(* CODESYS project bibliothek.library
   Company: er
   Title: er
   Placeholder: er
   Version: 0.0.1

Project tree, tasks and I/O mapping:
  libraries: GWP Library, * (Viessmann); Tc2_Standard, * (Beckhoff Automation GmbH); Tc2_System, * (Beckhoff Automation GmbH); Tc2_Utilities, * (Beckhoff Automation GmbH); Tc3_Module, * (Beckhoff Automation GmbH); VisuDialogs, * (System)
  DUTs/
    GVLs/
      global variables Globale_Uhr
  POUs/
    Funktionsblock/
    program MAIN [ST]
    program test [FBD]
  Version/
    global variables Global_Version
  VISUs/
    Alarmliste/
      visualisation Alarmliste
    Anlageseite_6/
      visualisation Kaeltekreis6_1
      visualisation Sollwertaenderung_C_6_3
      visualisation Zustandsanzeige
    Hauptmenu_3/
      visualisation Fusszeile_50
      visualisation Hauptmenu
      visualisation Kontaktseite3_1_50
      visualisation Uhr_einstellen3_1_50
    Home/
      visualisation Auswahlmenue
      visualisation Ein_Aus_Schalter
      visualisation Home_Standard_50
      visualisation RI_Schema_50
    IBN/
      visualisation IO_Auswahl
      visualisation Liste_AO
      visualisation Liste_DI
      visualisation SW_IBN_Einstellungen_K
    Infoseite/
      visualisation Infoliste
      visualisation Infoseite
    Sollwertmenu_9/
      Sollwertmenu/
        visualisation Sollwertmenu
      Wärmegewinnung/
        UWP/
          visualisation SW_Einstellungen_C
          visualisation SW_Einstellungen_DT
          visualisation SW_Einstellungen_K
          visualisation SW_Einstellungen_Zeit
          visualisation SW_WG_UWP_Verd
          visualisation SW_WG_UWP_Verd_Liste
        visualisation Sollwertmenu_Waermegewinnung
      Wärmepumpe/
      Wärmesenke/
      visualisation _SW_Heizgruppe
      visualisation _SW_Speicher_BWW
      visualisation _SW_Speicher_Heizung_1
      visualisation _SW_Speicher_Kaltwasser
      visualisation _SW_Waermegewinnung
      visualisation Sollwertmenu_Waermesenke
      visualisation SW_Waermepumpe
    Zeitprogramm/
      visualisation Wochenuhr_W7
    image pool Icon
    text list Sprachen
    visualisation test_1
  00000000-0000-0000-0000-000000000000|C:\Users\kuzr\Documents\Visual Studio 2013\Bildersammlung_VI\IC_102000\energietraeger_biomasse_fehler.png
  00000000-0000-0000-0000-000000000000|C:\Users\kuzr\Documents\Visual Studio 2013\Bildersammlung_VI\IC_102000\energietraeger_biomasse_inaktiv.png
  00000000-0000-0000-0000-000000000000|C:\Users\kuzr\Documents\Visual Studio 2013\Bildersammlung_VI\IC_102000\energietraeger_gas.png
  00000000-0000-0000-0000-000000000000|C:\Users\kuzr\Documents\Visual Studio 2013\Bildersammlung_VI\IC_102000\energietraeger_gas_fehler.png
  00000000-0000-0000-0000-000000000000|C:\Users\kuzr\Documents\Visual Studio 2013\Bildersammlung_VI\IC_102000\energietraeger_naturwaerme.png
  00000000-0000-0000-0000-000000000000|C:\Users\kuzr\Documents\Visual Studio 2013\Bildersammlung_VI\IC_102000\energietraeger_naturwaerme_fehler (2).png
  00000000-0000-0000-0000-000000000000|C:\Users\kuzr\Documents\Visual Studio 2013\Bildersammlung_VI\IC_102000\energietraeger_naturwaerme_fehler.png
  00000000-0000-0000-0000-000000000000|C:\Users\kuzr\Documents\Visual Studio 2013\Bildersammlung_VI\IC_102000\energietraeger_naturwaerme_inaktiv.png
  00000000-0000-0000-0000-000000000000|C:\Users\kuzr\Documents\Visual Studio 2013\Bildersammlung_VI\IC_102000\energietraeger_oel.png
  00000000-0000-0000-0000-000000000000|C:\Users\kuzr\Documents\Visual Studio 2013\Bildersammlung_VI\IC_102000\energietraeger_oel_inaktiv.png
  00000000-0000-0000-0000-000000000000|C:\Users\kuzr\Documents\Visual Studio 2013\Bildersammlung_VI\IC_102000\heizkreis_direkt (2).png
  00000000-0000-0000-0000-000000000000|C:\Users\kuzr\Documents\Visual Studio 2013\Bildersammlung_VI\IC_102000\heizkreis_direkt.png
  00000000-0000-0000-0000-000000000000|C:\Users\kuzr\Documents\Visual Studio 2013\Bildersammlung_VI\IC_102000\heizkreis_direkt_fehler.png
  00000000-0000-0000-0000-000000000000|C:\Users\kuzr\Documents\Visual Studio 2013\Bildersammlung_VI\IC_102000\heizkreis_direkt_inaktiv (2).png
  00000000-0000-0000-0000-000000000000|C:\Users\kuzr\Documents\Visual Studio 2013\Bildersammlung_VI\IC_102000\heizkreis_direkt_inaktiv.png
  00000000-0000-0000-0000-000000000000|C:\Users\kuzr\Documents\Visual Studio 2013\Bildersammlung_VI\IC_102000\heizkreis_fussbodenheizung.png
  00000000-0000-0000-0000-000000000000|C:\Users\kuzr\Documents\Visual Studio 2013\Bildersammlung_VI\IC_102000\heizkreis_fussbodenheizung_fehler.png
  00000000-0000-0000-0000-000000000000|C:\Users\kuzr\Documents\Visual Studio 2013\Bildersammlung_VI\IC_102000\heizkreis_fussbodenheizung_inaktiv.png
  00000000-0000-0000-0000-000000000000|C:\Users\kuzr\Documents\Visual Studio 2013\Bildersammlung_VI\IC_102000\heizkreis_mischer.png
  00000000-0000-0000-0000-000000000000|C:\Users\kuzr\Documents\Visual Studio 2013\Bildersammlung_VI\IC_102000\heizkreis_mischer_fehler.png
  00000000-0000-0000-0000-000000000000|C:\Users\kuzr\Documents\Visual Studio 2013\Bildersammlung_VI\IC_102000\heizkreis_mischer_inaktiv.png
  00000000-0000-0000-0000-000000000000|C:\Users\kuzr\Documents\Visual Studio 2013\Bildersammlung_VI\IC_102000\IC_102015_klappen_02.png
  00000000-0000-0000-0000-000000000000|C:\Users\kuzr\Documents\Visual Studio 2013\Bildersammlung_VI\IC_102000\klappen_01 (2).png
  00000000-0000-0000-0000-000000000000|C:\Users\kuzr\Documents\Visual Studio 2013\Bildersammlung_VI\IC_102000\klappen_01.png
  00000000-0000-0000-0000-000000000000|C:\Users\kuzr\Documents\Visual Studio 2013\Bildersammlung_VI\IC_102000\klappen_02.png
  00000000-0000-0000-0000-000000000000|C:\Users\kuzr\Documents\Visual Studio 2013\Bildersammlung_VI\IC_102000\komponente_detail_heizkreis.png
  00000000-0000-0000-0000-000000000000|C:\Users\kuzr\Documents\Visual Studio 2013\Bildersammlung_VI\IC_102000\komponente_detail_klappe (2).png
  00000000-0000-0000-0000-000000000000|C:\Users\kuzr\Documents\Visual Studio 2013\Bildersammlung_VI\IC_102000\komponente_detail_klappe.png
  00000000-0000-0000-0000-000000000000|C:\Users\kuzr\Documents\Visual Studio 2013\Bildersammlung_VI\IC_102000\komponente_detail_klappe_fehler (2).png
  00000000-0000-0000-0000-000000000000|C:\Users\kuzr\Documents\Visual Studio 2013\Bildersammlung_VI\IC_102000\komponente_detail_klappe_fehler.png
  00000000-0000-0000-0000-000000000000|C:\Users\kuzr\Documents\Visual Studio 2013\Bildersammlung_VI\IC_102000\komponente_detail_klappe_inaktiv.png
  00000000-0000-0000-0000-000000000000|C:\Users\kuzr\Documents\Visual Studio 2013\Bildersammlung_VI\IC_102000\komponente_detail_klappe_inaktiv_2.png
  00000000-0000-0000-0000-000000000000|C:\Users\kuzr\Documents\Visual Studio 2013\Bildersammlung_VI\IC_102000\komponente_detail_mischer_01.png
  00000000-0000-0000-0000-000000000000|C:\Users\kuzr\Documents\Visual Studio 2013\Bildersammlung_VI\IC_102000\komponente_detail_mischer_02.png
  00000000-0000-0000-0000-000000000000|C:\Users\kuzr\Documents\Visual Studio 2013\Bildersammlung_VI\IC_102000\komponente_detail_mischer_fehler.png
  00000000-0000-0000-0000-000000000000|C:\Users\kuzr\Documents\Visual Studio 2013\Bildersammlung_VI\IC_102000\komponente_detail_mischer_inaktiv.png
  00000000-0000-0000-0000-000000000000|C:\Users\kuzr\Documents\Visual Studio 2013\Bildersammlung_VI\IC_102000\komponente_detail_pumpe.png
  00000000-0000-0000-0000-000000000000|C:\Users\kuzr\Documents\Visual Studio 2013\Bildersammlung_VI\IC_102000\komponente_detail_pumpe_fehler.png
  00000000-0000-0000-0000-000000000000|C:\Users\kuzr\Documents\Visual Studio 2013\Bildersammlung_VI\IC_102000\komponente_detail_pumpe_inaktiv.png
  00000000-0000-0000-0000-000000000000|C:\Users\kuzr\Documents\Visual Studio 2013\Bildersammlung_VI\IC_102000\mischer_01.png
  00000000-0000-0000-0000-000000000000|C:\Users\kuzr\Documents\Visual Studio 2013\Bildersammlung_VI\IC_102000\mischer_02.png
  00000000-0000-0000-0000-000000000000|C:\Users\kuzr\Documents\Visual Studio 2013\Bildersammlung_VI\IC_102000\mischer_03.png
  00000000-0000-0000-0000-000000000000|C:\Users\kuzr\Documents\Visual Studio 2013\Bildersammlung_VI\IC_102000\mischer_04.png
  00000000-0000-0000-0000-000000000000|C:\Users\kuzr\Documents\Visual Studio 2013\Bildersammlung_VI\IC_102000\mischer_05.png
  00000000-0000-0000-0000-000000000000|C:\Users\kuzr\Documents\Visual Studio 2013\Bildersammlung_VI\IC_102000\mischer_06.png
  00000000-0000-0000-0000-000000000000|C:\Users\kuzr\Documents\Visual Studio 2013\Bildersammlung_VI\IC_102000\mischer_07.png
  00000000-0000-0000-0000-000000000000|C:\Users\kuzr\Documents\Visual Studio 2013\Bildersammlung_VI\IC_102000\mischer_08.png
  00000000-0000-0000-0000-000000000000|C:\Users\kuzr\Documents\Visual Studio 2013\Bildersammlung_VI\IC_102000\mischer_09.png
  00000000-0000-0000-0000-000000000000|C:\Users\kuzr\Documents\Visual Studio 2013\Bildersammlung_VI\IC_102000\mischer_10.png
  00000000-0000-0000-0000-000000000000|C:\Users\kuzr\Documents\Visual Studio 2013\Bildersammlung_VI\IC_102000\mischer_11.png
  00000000-0000-0000-0000-000000000000|C:\Users\kuzr\Documents\Visual Studio 2013\Bildersammlung_VI\IC_102000\mischer_12.png
  00000000-0000-0000-0000-000000000000|C:\Users\kuzr\Documents\Visual Studio 2013\Bildersammlung_VI\IC_102000\pumpe_links.png
  00000000-0000-0000-0000-000000000000|C:\Users\kuzr\Documents\Visual Studio 2013\Bildersammlung_VI\IC_102000\pumpe_oben.png
  00000000-0000-0000-0000-000000000000|C:\Users\kuzr\Documents\Visual Studio 2013\Bildersammlung_VI\IC_102000\pumpe_rechts.png
  00000000-0000-0000-0000-000000000000|C:\Users\kuzr\Documents\Visual Studio 2013\Bildersammlung_VI\IC_102000\pumpe_unten.png
  00000000-0000-0000-0000-000000000000|C:\Users\kuzr\Documents\Visual Studio 2013\Bildersammlung_VI\IC_102000\speicher_eis.png
  00000000-0000-0000-0000-000000000000|C:\Users\kuzr\Documents\Visual Studio 2013\Bildersammlung_VI\IC_102000\speicher_eis_fehler.png
  00000000-0000-0000-0000-000000000000|C:\Users\kuzr\Documents\Visual Studio 2013\Bildersammlung_VI\IC_102000\speicher_eis_inaktiv.png
  00000000-0000-0000-0000-000000000000|C:\Users\kuzr\Documents\Visual Studio 2013\Bildersammlung_VI\IC_102000\speicher_heizen.png
  00000000-0000-0000-0000-000000000000|C:\Users\kuzr\Documents\Visual Studio 2013\Bildersammlung_VI\IC_102000\speicher_heizen_fehler.png
  00000000-0000-0000-0000-000000000000|C:\Users\kuzr\Documents\Visual Studio 2013\Bildersammlung_VI\IC_102000\speicher_heizen_inaktiv.png
  00000000-0000-0000-0000-000000000000|C:\Users\kuzr\Documents\Visual Studio 2013\Bildersammlung_VI\IC_102000\speicher_warmwasser.png
  00000000-0000-0000-0000-000000000000|C:\Users\kuzr\Documents\Visual Studio 2013\Bildersammlung_VI\IC_102000\speicher_warmwasser_fehler.png
  00000000-0000-0000-0000-000000000000|C:\Users\kuzr\Documents\Visual Studio 2013\Bildersammlung_VI\IC_102000\speicher_warmwasser_inaktiv.png
  00000000-0000-0000-0000-000000000000|C:\Users\kuzr\Documents\Visual Studio 2013\Bildersammlung_VI\IC_102000\energietraeger_biomasse.png
  00000000-0000-0000-0000-000000000000|C:\Users\kuzr\Documents\Visual Studio 2013\Bildersammlung_VI\IC_106000\komponente_brenner.png
  00000000-0000-0000-0000-000000000000|C:\Users\kuzr\Documents\Visual Studio 2013\Bildersammlung_VI\IC_106000\komponente_brenner_fehler.png
  00000000-0000-0000-0000-000000000000|C:\Users\kuzr\Documents\Visual Studio 2013\Bildersammlung_VI\IC_106000\komponente_brenner_inaktiv.png
  00000000-0000-0000-0000-000000000000|C:\Users\kuzr\Documents\Visual Studio 2013\Bildersammlung_VI\IC_106000\speicher.png
  00000000-0000-0000-0000-000000000000|C:\Users\kuzr\Documents\Visual Studio 2013\Bildersammlung_VI\IC_106000\speicher_eis.png
  00000000-0000-0000-0000-000000000000|C:\Users\kuzr\Documents\Visual Studio 2013\Bildersammlung_VI\IC_106000\system_leistung_nicht_touchbar.png
  00000000-0000-0000-0000-000000000000|C:\Users\kuzr\Documents\Visual Studio 2013\Bildersammlung_VI\IC_106000\system_leistung_touchbar.png
  00000000-0000-0000-0000-000000000000|C:\Users\kuzr\Documents\Visual Studio 2013\Bildersammlung_VI\IC_106000\waermetauscher.png
  00000000-0000-0000-0000-000000000000|C:\Users\kuzr\Documents\Visual Studio 2013\Bildersammlung_VI\IC_106000\weiche.png
  00000000-0000-0000-0000-000000000000|C:\Users\kuzr\Documents\Visual Studio 2013\Bildersammlung_VI\IC_108000\komponente_brenner_fehler.png
  00000000-0000-0000-0000-000000000000|C:\Users\kuzr\Documents\Visual Studio 2013\Bildersammlung_VI\IC_108000\komponente_brenner_inaktiv.png
  00000000-0000-0000-0000-000000000000|C:\Users\kuzr\Documents\Visual Studio 2013\Bildersammlung_VI\IC_108000\speicher.png
  00000000-0000-0000-0000-000000000000|C:\Users\kuzr\Documents\Visual Studio 2013\Bildersammlung_VI\IC_108000\speicher_eis.png
  00000000-0000-0000-0000-000000000000|C:\Users\kuzr\Documents\Visual Studio 2013\Bildersammlung_VI\IC_108000\komponente_brenner.png
  00000000-0000-0000-0000-000000000000|C:\Users\kuzr\Documents\Visual Studio 2013\Bildersammlung_VI\IC_111000\bildschirm_reinigen.png
  00000000-0000-0000-0000-000000000000|C:\Users\kuzr\Documents\Visual Studio 2013\Bildersammlung_VI\IC_111000\dokumentation.png
  00000000-0000-0000-0000-000000000000|C:\Users\kuzr\Documents\Visual Studio 2013\Bildersammlung_VI\IC_111000\kontaktdaten_nutzer.png
  00000000-0000-0000-0000-000000000000|C:\Users\kuzr\Documents\Visual Studio 2013\Bildersammlung_VI\IC_111000\kontaktdaten_viessmann.png
  00000000-0000-0000-0000-000000000000|C:\Users\kuzr\Documents\Visual Studio 2013\Bildersammlung_VI\IC_111000\nutzeranmeldung.png
  00000000-0000-0000-0000-000000000000|C:\Users\kuzr\Documents\Visual Studio 2013\Bildersammlung_VI\IC_111000\oberflaeche_schließen.png
  00000000-0000-0000-0000-000000000000|C:\Users\kuzr\Documents\Visual Studio 2013\Bildersammlung_VI\IC_111000\pruefbetrieb.png
  00000000-0000-0000-0000-000000000000|C:\Users\kuzr\Documents\Visual Studio 2013\Bildersammlung_VI\IC_111000\system_konfigurieren.png
  00000000-0000-0000-0000-000000000000|C:\Users\kuzr\Documents\Visual Studio 2013\Bildersammlung_VI\IC_111000\betriebszaehler_zuruecksetzen.png
  00000000-0000-0000-0000-000000000000|C:\Users\kuzr\Documents\Visual Studio 2013\Bildersammlung_VI\IC_112000\abschaltbetrieb.png
  00000000-0000-0000-0000-000000000000|C:\Users\kuzr\Documents\Visual Studio 2013\Bildersammlung_VI\IC_112000\aktiv.png
  00000000-0000-0000-0000-000000000000|C:\Users\kuzr\Documents\Visual Studio 2013\Bildersammlung_VI\IC_112000\an.png
  00000000-0000-0000-0000-000000000000|C:\Users\kuzr\Documents\Visual Studio 2013\Bildersammlung_VI\IC_112000\astatur_01.png
  00000000-0000-0000-0000-000000000000|C:\Users\kuzr\Documents\Visual Studio 2013\Bildersammlung_VI\IC_112000\auf.png
  00000000-0000-0000-0000-000000000000|C:\Users\kuzr\Documents\Visual Studio 2013\Bildersammlung_VI\IC_112000\aus.png
  00000000-0000-0000-0000-000000000000|C:\Users\kuzr\Documents\Visual Studio 2013\Bildersammlung_VI\IC_112000\bedingung_erfuellt.png
  00000000-0000-0000-0000-000000000000|C:\Users\kuzr\Documents\Visual Studio 2013\Bildersammlung_VI\IC_112000\bedingung_nicht_erfuellt.png
  00000000-0000-0000-0000-000000000000|C:\Users\kuzr\Documents\Visual Studio 2013\Bildersammlung_VI\IC_112000\email_prueftaste.png
  00000000-0000-0000-0000-000000000000|C:\Users\kuzr\Documents\Visual Studio 2013\Bildersammlung_VI\IC_112000\erfuellt.png
  00000000-0000-0000-0000-000000000000|C:\Users\kuzr\Documents\Visual Studio 2013\Bildersammlung_VI\IC_112000\exportieren.png
  00000000-0000-0000-0000-000000000000|C:\Users\kuzr\Documents\Visual Studio 2013\Bildersammlung_VI\IC_112000\frostschutzbetrieb.png
  00000000-0000-0000-0000-000000000000|C:\Users\kuzr\Documents\Visual Studio 2013\Bildersammlung_VI\IC_112000\haeckchen_ungesetzt (2).png
  00000000-0000-0000-0000-000000000000|C:\Users\kuzr\Documents\Visual Studio 2013\Bildersammlung_VI\IC_112000\haeckchen_ungesetzt.png
  00000000-0000-0000-0000-000000000000|C:\Users\kuzr\Documents\Visual Studio 2013\Bildersammlung_VI\IC_112000\home.png
  00000000-0000-0000-0000-000000000000|C:\Users\kuzr\Documents\Visual Studio 2013\Bildersammlung_VI\IC_112000\home_uebersicht.png
  00000000-0000-0000-0000-000000000000|C:\Users\kuzr\Documents\Visual Studio 2013\Bildersammlung_VI\IC_112000\inaktiv.png
  00000000-0000-0000-0000-000000000000|C:\Users\kuzr\Documents\Visual Studio 2013\Bildersammlung_VI\IC_112000\intervall.png
  00000000-0000-0000-0000-000000000000|C:\Users\kuzr\Documents\Visual Studio 2013\Bildersammlung_VI\IC_112000\Itastatur_03.png
  00000000-0000-0000-0000-000000000000|C:\Users\kuzr\Documents\Visual Studio 2013\Bildersammlung_VI\IC_112000\ja.png
  00000000-0000-0000-0000-000000000000|C:\Users\kuzr\Documents\Visual Studio 2013\Bildersammlung_VI\IC_112000\kopieren.png
  00000000-0000-0000-0000-000000000000|C:\Users\kuzr\Documents\Visual Studio 2013\Bildersammlung_VI\IC_112000\laden.png
  00000000-0000-0000-0000-000000000000|C:\Users\kuzr\Documents\Visual Studio 2013\Bildersammlung_VI\IC_112000\listenansicht.png
  00000000-0000-0000-0000-000000000000|C:\Users\kuzr\Documents\Visual Studio 2013\Bildersammlung_VI\IC_112000\meldelisten_archiv.png
  00000000-0000-0000-0000-000000000000|C:\Users\kuzr\Documents\Visual Studio 2013\Bildersammlung_VI\IC_112000\meldelisten_einstellungen.png
  00000000-0000-0000-0000-000000000000|C:\Users\kuzr\Documents\Visual Studio 2013\Bildersammlung_VI\IC_112000\meldungen_weiterleiten.png
  00000000-0000-0000-0000-000000000000|C:\Users\kuzr\Documents\Visual Studio 2013\Bildersammlung_VI\IC_112000\menue.png
  00000000-0000-0000-0000-000000000000|C:\Users\kuzr\Documents\Visual Studio 2013\Bildersammlung_VI\IC_112000\minus.png
  00000000-0000-0000-0000-000000000000|C:\Users\kuzr\Documents\Visual Studio 2013\Bildersammlung_VI\IC_112000\nein.png
  00000000-0000-0000-0000-000000000000|C:\Users\kuzr\Documents\Visual Studio 2013\Bildersammlung_VI\IC_112000\nicht_erfuellt.png
  00000000-0000-0000-0000-000000000000|C:\Users\kuzr\Documents\Visual Studio 2013\Bildersammlung_VI\IC_112000\normalbetrieb.png
  00000000-0000-0000-0000-000000000000|C:\Users\kuzr\Documents\Visual Studio 2013\Bildersammlung_VI\IC_112000\pfeil_rechts.png
  00000000-0000-0000-0000-000000000000|C:\Users\kuzr\Documents\Visual Studio 2013\Bildersammlung_VI\IC_112000\plus.png
  00000000-0000-0000-0000-000000000000|C:\Users\kuzr\Documents\Visual Studio 2013\Bildersammlung_VI\IC_112000\quittieren_aus.png
  00000000-0000-0000-0000-000000000000|C:\Users\kuzr\Documents\Visual Studio 2013\Bildersammlung_VI\IC_112000\quittierena_an.png
  00000000-0000-0000-0000-000000000000|C:\Users\kuzr\Documents\Visual Studio 2013\Bildersammlung_VI\IC_112000\radiobutton_gesetzt.png
  00000000-0000-0000-0000-000000000000|C:\Users\kuzr\Documents\Visual Studio 2013\Bildersammlung_VI\IC_112000\radiobutton_ungesetzt.png
  text list GlobalTextList
*)

// DUTs/GVLs/Globale_Uhr
{attribute 'qualified_only'}
VAR_GLOBAL
	
	   systemtimestruct		: timestruct;   
END_VAR

// Version/Global_Version
{attribute 'TcGenerated'}
// This function has been automatically generated from the project information.
VAR_GLOBAL CONSTANT
	{attribute 'const_non_replaced'}
	{attribute 'linkalways'}
	stLibVersion_er : ST_LibVersion := (iMajor := 0, iMinor := 0, iBuild := 1, iRevision := 0, sVersion := '0.0.1');
END_VAR

// POUs/MAIN
PROGRAM MAIN
VAR

	

END_VAR

END_PROGRAM

// POUs/test
PROGRAM test
VAR

	
	Globale_Zeit_0: Globale_Zeit;
    CLK_W_0: CLK_W;
	
	GR_2_0: GR_2;
	
	


	CLK_W7_0: CLK_W7;
	Logger_0: Logger;
	GR_4_mit_RE_0: GR_4_mit_RE;
END_VAR

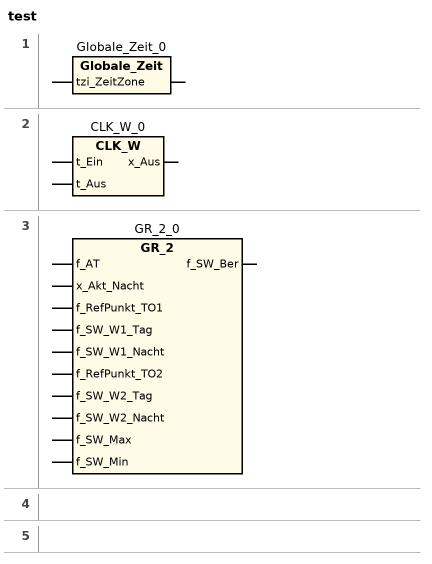
// NETWORK 1
Globale_Zeit_0(); // Globale_Zeit

// NETWORK 2
CLK_W_0(); // CLK_W

// NETWORK 3
GR_2_0(); // GR_2

// NETWORK 4

// NETWORK 5

END_PROGRAM

// VISUs/Alarmliste/Alarmliste
VISUALIZATION Alarmliste  // 800x430
END_VISUALIZATION

// VISUs/Anlageseite_6/Kaeltekreis6_1
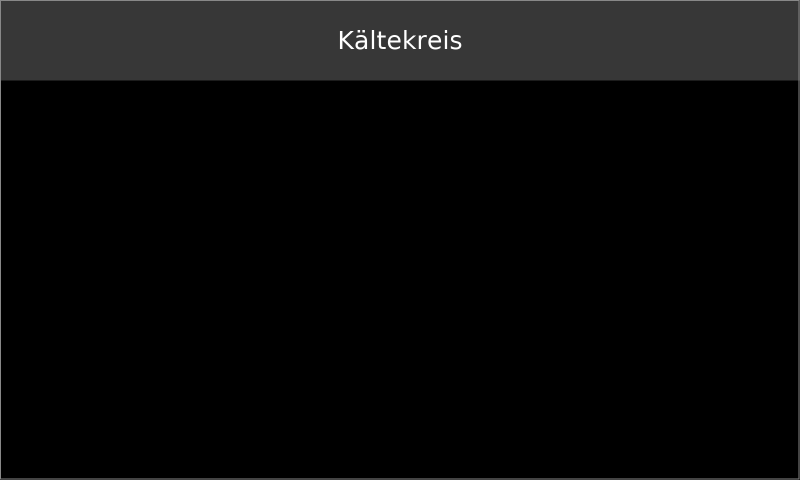
VISUALIZATION Kaeltekreis6_1  // 800x480
    Rectangle (0,0 800x80), "Kältekreis"
END_VISUALIZATION

// VISUs/Anlageseite_6/Sollwertaenderung_C_6_3
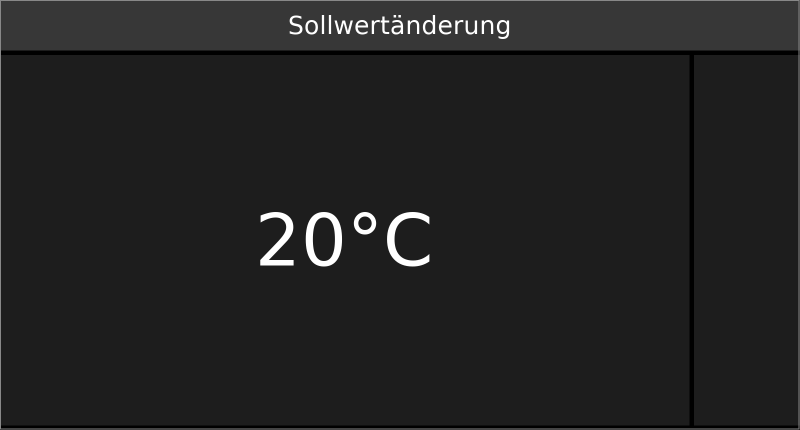
VISUALIZATION Sollwertaenderung_C_6_3  // 800x430
    Rectangle (0,0 800x50), "Sollwertänderung"
    Rectangle (0,55 689x370), "20°C"
    Rectangle (694,55 106x370)
END_VISUALIZATION

// VISUs/Anlageseite_6/Zustandsanzeige
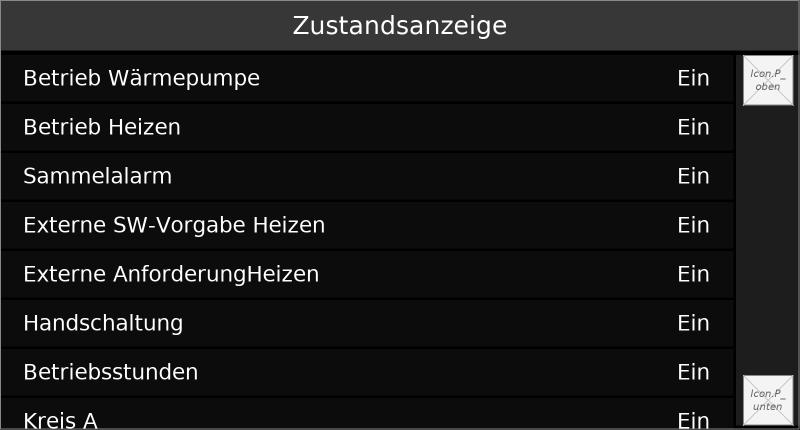
VISUALIZATION Zustandsanzeige  // 800x430
VAR_IN_OUT
	auf:BOOL;
		
END_VAR
    Image (1113,281 30x116), image: Icon.waermetauscher
    Group (0,0 800x640)
        Rectangle (0,0 800x50), "Zustandsanzeige"
        Group (0,430 800x50)
            Rectangle (0,0 800x50)
            Image (25,0 50x50), image: Icon.home
            Image (425,0 50x50), image: Icon.reinnavigieren
            Image (625,0 50x50), image: Icon.warnung_rot
            Image (125,0 50x50), image: Icon.zurueck
            Image (325,0 50x50), image: Icon.reinnavigieren
            Image (325,0 50x50), image: Icon.p_links
            Image (425,0 50x50), image: Icon.P_rechts
        Rectangle (0,55 733x46)
        Label (20,55 479x46), "Betrieb Wärmepumpe"
        Rectangle (0,104 733x46)
        Label (20,104 479x46), "Betrieb Heizen"
        Rectangle (0,153 733x46)
        Label (20,153 479x46), "Sammelalarm"
        Rectangle (0,202 733x46)
        Label (20,202 479x46), "Externe SW-Vorgabe Heizen"
        Rectangle (0,251 733x46)
        Label (20,251 479x46), "Externe AnforderungHeizen"
        Rectangle (0,300 733x46)
        Label (20,300 479x46), "Handschaltung"
        Rectangle (0,349 733x46)
        Label (20,349 479x46), "Betriebsstunden"
        Rectangle (583,55 130x46), "Ein"
        Rectangle (583,104 130x46), "Ein"
        Rectangle (0,398 733x46)
        Label (20,398 479x46), "Kreis A"
        Rectangle (0,447 733x46)
        Label (20,447 479x46), "Kreis B"
        Rectangle (0,496 733x46)
        Label (20,496 479x46), "Stufe 1"
        Rectangle (0,545 733x46)
        Label (20,545 479x46), "Stufe 2"
        Rectangle (583,545 130x46), "Ein"
        Rectangle (0,594 733x46)
        Label (20,594 479x46), "Stufe 3"
        Rectangle (583,153 130x46), "Ein"
        Rectangle (583,202 130x46), "Ein"
        Rectangle (583,251 130x46), "Ein"
        Rectangle (583,349 130x46), "Ein"
        Rectangle (583,300 130x46), "Ein"
        Rectangle (583,398 130x46), "Ein"
        Rectangle (583,447 130x46), "Ein"
        Rectangle (583,496 130x46), "Ein"
        Rectangle (583,594 130x46), "Ein"
        Rectangle (736,55 64x370)
        Image (743,55 50x50), image: Icon.P_oben
            OnMouseClick: write the text variable via Default
        Image (743,375 50x50), image: Icon.P_unten
END_VISUALIZATION

// VISUs/Hauptmenu_3/Fusszeile_50
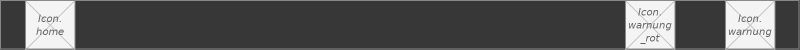
VISUALIZATION Fusszeile_50  // 800x50
    Group (0,0 800x50)
        Rectangle (0,0 800x50)
        Image (625,0 50x50), image: Icon.warnung_rot
            OnMouseClick: execute { GWP_Library.Visu.i_Frame_Index:=0; }
        Image (25,0 50x50), image: Icon.home
            OnMouseClick:  Assign=Home_Standard_50, Type=Assignment
            OnMouseClick: execute { GWP_Library.Visu.i_Frame_Index:=0; }
        Image (725,0 50x50), image: Icon.warnung
            OnMouseClick:  Assign=Infoseite, Type=Assignment
            OnMouseClick: execute { GWP_Library.Visu.i_Frame_Index:=0; }
END_VISUALIZATION

// VISUs/Hauptmenu_3/Hauptmenu
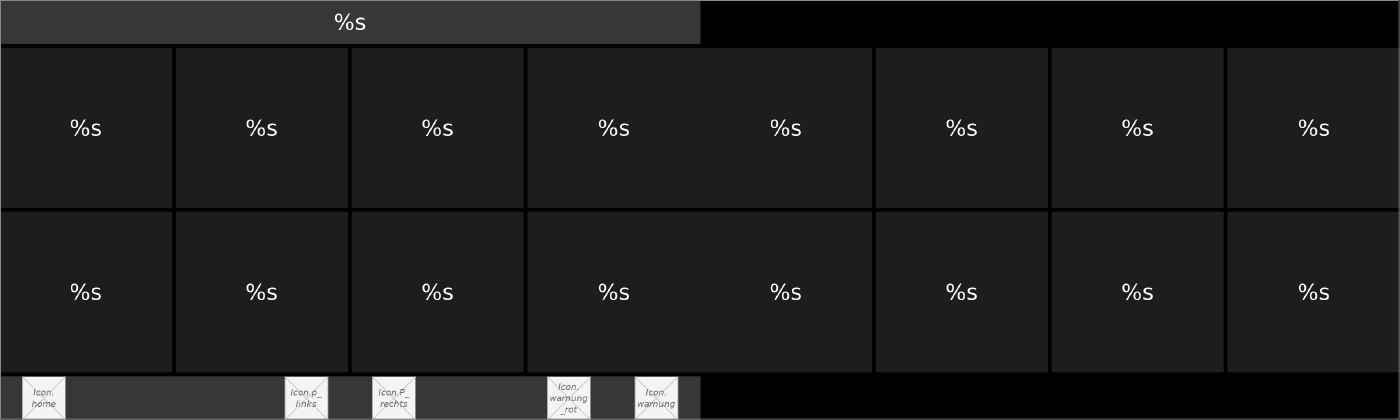
VISUALIZATION Hauptmenu  // 1600x480
VAR_IN_OUT
		
END_VAR

VAR
	i_verschieben:INT;

END_VAR
    Image (425,430 50x50), image: Icon.reinnavigieren
    Image (325,430 50x50), image: Icon.reinnavigieren
    Rectangle (0,0 800x50), "%s", text list: 'Sprachen', text index: 32
    Frame (0,430 800x50)
        shows Fusszeile_50()
    Group (0,55 1600x370)
        p3560616238: i_verschieben
        Rectangle (0,0 196x182), "%s", text list: 'Sprachen', text index: 33
        Rectangle (201,0 196x182), "%s", text list: 'Sprachen', text index: 34
        Rectangle (402,0 196x182), "%s", text list: 'Sprachen', text index: 35
            OnMouseClick:  Assign=Sollwertmenu, Type=Assignment
        Rectangle (603,0 197x182), "%s", text list: 'Sprachen', text index: 36
        Rectangle (0,187 196x183), "%s", text list: 'Sprachen', text index: 37
            OnMouseClick:  Assign=Uhr_einstellen3_1_50, Type=Assignment
        Rectangle (201,187 196x183), "%s", text list: 'Sprachen', text index: 38
            OnMouseClick:  Assign=IO_Auswahl, Type=Assignment
        Rectangle (402,187 196x183), "%s", text list: 'Sprachen', text index: 39
        Rectangle (603,187 197x183), "%s", text list: 'Sprachen', text index: 40
            OnMouseClick:  Assign=Kontaktseite3_1_50, Type=Assignment
        Rectangle (800,0 196x182), "%s"
        Rectangle (1001,0 196x182), "%s"
        Rectangle (1202,0 196x182), "%s"
            OnMouseClick:  Assign=Sollwertmenu, Type=Assignment
        Rectangle (1403,0 197x182), "%s"
        Rectangle (800,187 196x183), "%s"
            OnMouseClick:  Assign=Uhr_einstellen3_1_50, Type=Assignment
        Rectangle (1001,187 196x183), "%s"
            OnMouseClick:  Assign=IO_Auswahl, Type=Assignment
        Rectangle (1202,187 196x183), "%s"
        Rectangle (1403,187 197x183), "%s"
            OnMouseClick:  Assign=Kontaktseite3_1_50, Type=Assignment
    Image (425,430 50x50), image: Icon.P_rechts
        OnMouseClick: execute {
            IF i_verschieben>-800 THEN
            	i_verschieben:=i_verschieben-800;
            END_IF
        }
    Image (325,430 50x50), image: Icon.p_links
        OnMouseClick: execute {
            IF i_verschieben<0 THEN
            	i_verschieben:=i_verschieben+800;
            END_IF
        }
END_VISUALIZATION

// VISUs/Hauptmenu_3/Kontaktseite3_1_50
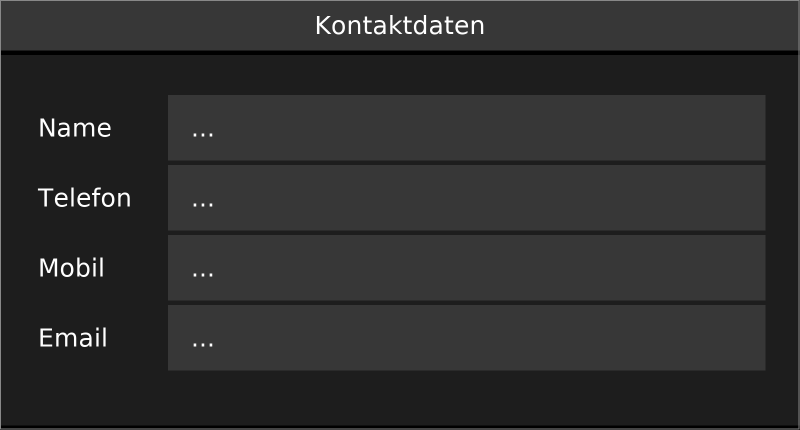
VISUALIZATION Kontaktseite3_1_50  // 800x430
    Rectangle (0,0 800x50), "Kontaktdaten"
    Rectangle (0,55 800x370)
    Rectangle (168,95 597x65)
    Rectangle (168,165 597x65)
    Rectangle (168,235 597x65)
    Rectangle (168,305 597x65)
    Label (35,95 113x65), "Name"
    Label (35,165 113x65), "Telefon"
    Label (35,235 113x65), "Mobil"
    Label (35,305 113x65), "Email"
    Label (188,305 557x65), "..."
    Label (188,235 557x65), "..."
    Label (188,165 557x65), "..."
    Label (188,95 557x65), "..."
    Frame (0,430 800x50)
        shows Fusszeile_50()
END_VISUALIZATION

// VISUs/Hauptmenu_3/Uhr_einstellen3_1_50
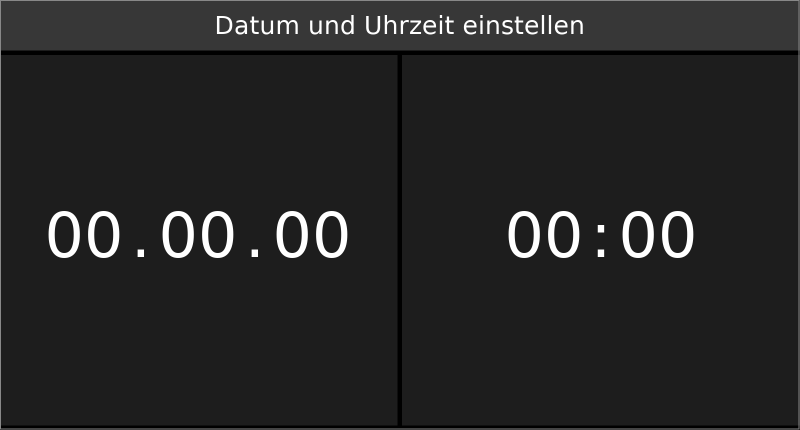
VISUALIZATION Uhr_einstellen3_1_50  // 800x430
    Frame (0,430 800x50)
        shows Fusszeile_50()
    Rectangle (0,0 800x50), "Datum und Uhrzeit einstellen"
    Rectangle (0,55 397x370)
    Rectangle (402,55 398x370)
    Image (425,430 50x50), image: Icon.reinnavigieren
    Image (125,430 50x50), image: Icon.zurueck
        OnMouseClick:  Assign=Hauptmenu, Type=Assignment
    Image (325,430 50x50), image: Icon.reinnavigieren
    Group (502,193 198x84)
        Rectangle (84,0 30x84), ":"
        Rectangle (0,0 84x84), "00"
        Rectangle (114,0 84x84), "00"
    Rectangle (156,193 84x84), "00"
    Rectangle (126,193 30x84), "."
    Rectangle (42,193 84x84), "00"
    Rectangle (240,193 30x84), "."
    Rectangle (270,193 84x84), "00"
END_VISUALIZATION

// VISUs/Home/Auswahlmenue
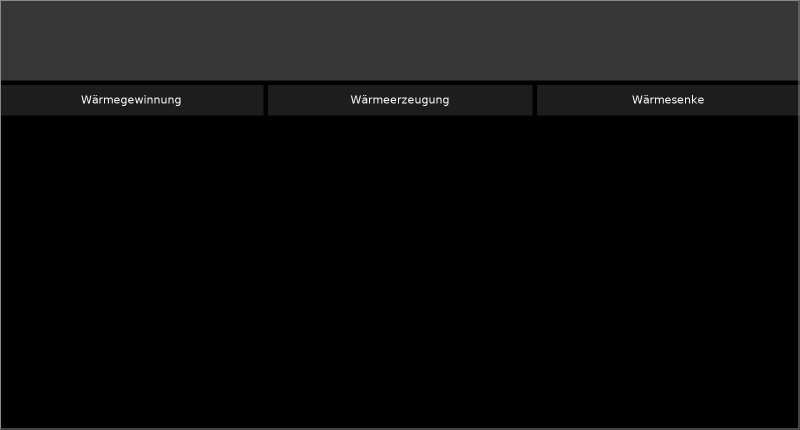
VISUALIZATION Auswahlmenue  // 800x430
    Rectangle (0,0 800x80)
    Rectangle (0,85 263x30), "Wärmegewinnung"
    Rectangle (268,85 264x30), "Wärmeerzeugung"
    Rectangle (537,85 263x30), "Wärmesenke"
END_VISUALIZATION

// VISUs/Home/Ein_Aus_Schalter
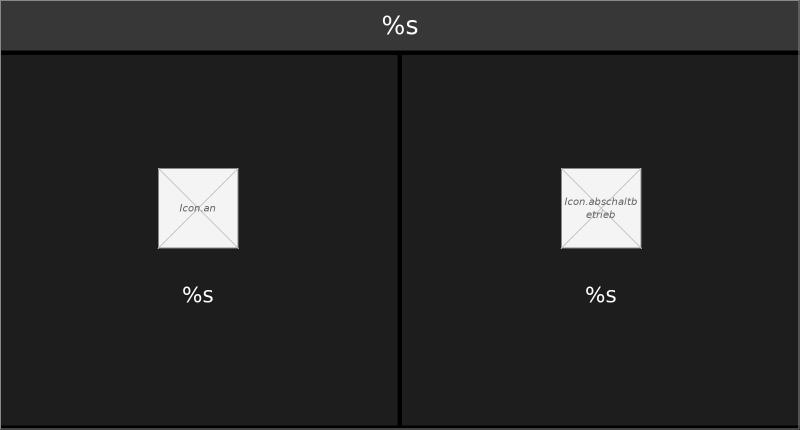
VISUALIZATION Ein_Aus_Schalter  // 800x430
VAR_IN_OUT
	x_Status:BOOL;
	i_Status:INT:=i_Text_2;
END_VAR

VAR_OUTPUT
	
	
END_VAR

VAR_INPUT
	i_Titel:INT;
	i_Text_1:INT;
	i_Text_2:INT;	
END_VAR
    Rectangle (0,0 800x50), "%s", text list: 'Sprachen', text index: i_Titel
    Rectangle (0,55 397x370)
    Rectangle (0,55 397x5)
    Image (158,168 80x80), image: Icon.an
    Rectangle (123,280 150x30), "%s", text list: 'Sprachen', text index: i_Text_1
        OnMouseClick: execute { x_Status:=TRUE; i_Status:=i_Text_1; }
    Image (125,430 50x50), image: Icon.zurueck
        OnMouseClick: execute { GWP_Library.Visu.i_Frame_Index:=0; }
    Rectangle (402,55 398x370)
    Rectangle (402,55 398x5)
    Rectangle (526,280 150x30), "%s", text list: 'Sprachen', text index: i_Text_2
        OnMouseClick: execute { x_Status:=FALSE; i_Status:=i_Text_2; }
    Image (561,168 80x80), image: Icon.abschaltbetrieb
    Polygon (943,131)
END_VISUALIZATION

// VISUs/Home/Home_Standard_50
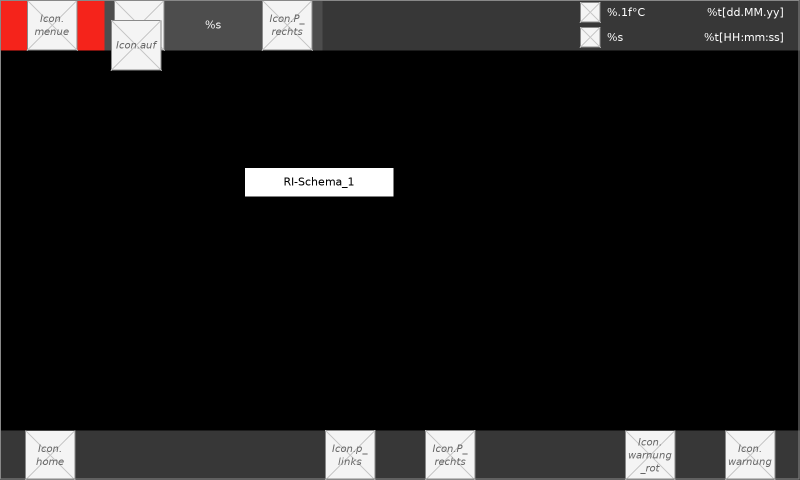
VISUALIZATION Home_Standard_50  // 800x480
VAR_IN_OUT

END_VAR

VAR
	i_Anzeige:INT;	
	x_Temp:BOOL;
	
END_VAR
    Frame (0,430 800x50)
        shows Fusszeile_50()
    Frame (0,0 800x430), frame switch variable: GWP_Library.Visu.i_Frame_Index
        shows RI_Schema_50(i_Status := i_Anzeige)
        shows Ein_Aus_Schalter(i_Titel := 41, i_Text_1 := 42, i_Text_2 := 43, x_Status := x_Temp, i_Status := i_Anzeige)
END_VISUALIZATION

// VISUs/Home/RI_Schema_50
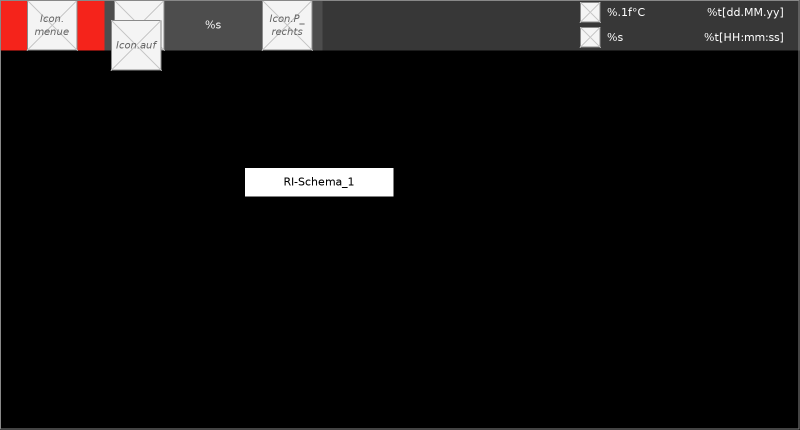
VISUALIZATION RI_Schema_50  // 800x430
VAR
	i_verschieben:INT;
	
END_VAR

VAR_INPUT
	i_Status:INT;
	
END_VAR
    Rectangle (0,0 800x50)
    Rectangle (702,0 85x25), "%t[dd.MM.yy]"
    Rectangle (702,25 85x25), "%t[HH:mm:ss]"
    Image (580,27 20x20), image: Icon.login_status
    Rectangle (604,0 85x25), "%.1f°C"
    Rectangle (604,25 85x25), "%s"
    Rectangle (104,0 218x50), "%s", text list: 'Sprachen', text index: i_Status
        OnMouseClick: execute { GWP_Library.Visu.i_Frame_Index:=1; }
    Image (114,0 50x50), image: Icon.an
    Rectangle (0,0 104x50)
        OnMouseClick:  Assign=Hauptmenu, Type=Assignment
    Image (27,0 50x50), image: Icon.menue
        OnMouseClick:  Assign=Hauptmenu, Type=Assignment
    Image (425,430 50x50), image: Icon.P_rechts
        OnMouseClick: execute {
            IF i_verschieben>-800 THEN
            	i_verschieben:=i_verschieben-400;
            END_IF
        }
    Image (325,430 50x50), image: Icon.p_links
        OnMouseClick: execute {
            IF i_verschieben<0 THEN
            	i_verschieben:=i_verschieben+400;
            END_IF
        }
    Image (580,2 20x20), image: Icon.aussentemperatur
    Image (262,0 50x50), image: Icon.P_rechts
    Group (244,167 848x88)
        p3560616238: i_verschieben
        Rectangle (0,0 150x30), "RI-Schema_1"
        Rectangle (698,58 150x30), "RI-Schema_2"
    Image (111,20 50x50), image: Icon.auf
END_VISUALIZATION

// VISUs/IBN/IO_Auswahl
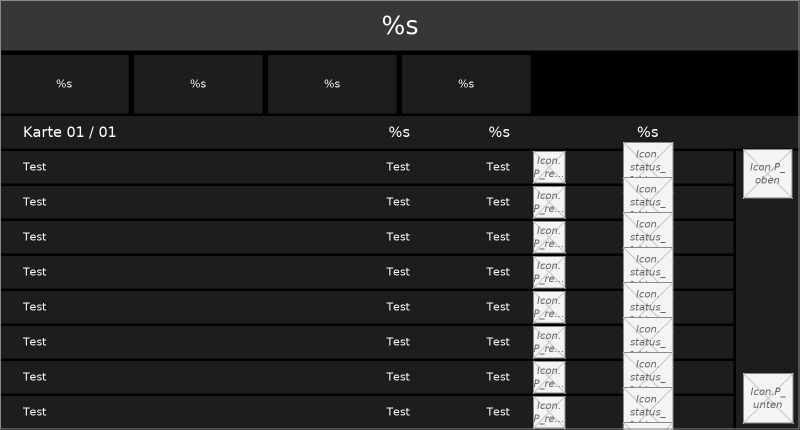
VISUALIZATION IO_Auswahl  // 800x430
    Rectangle (0,0 800x50), "%s", text list: 'Sprachen', text index: 44
    Rectangle (0,55 128x58), "%s", text list: 'Sprachen', text index: 45
        OnMouseClick: FrameSelectionChange Selection=SelectedFrame=bf6d0b13-4f63-4973-a15e-614a474f48dd, Selection=1, GlobSel=AssignType=Directly, SelType=Locally
    Rectangle (134,55 128x58), "%s", text list: 'Sprachen', text index: 46
        OnMouseClick: execute { GWP_Library.Visu.i_Frame_Index:=1; }
    Rectangle (268,55 128x58), "%s", text list: 'Sprachen', text index: 47
    Rectangle (402,55 128x58), "%s", text list: 'Sprachen', text index: 48
    Rectangle (0,55 128x5)
    Rectangle (134,55 128x5)
    Rectangle (268,55 128x5)
    Rectangle (402,55 128x5)
    Frame (0,116 800x279)
        shows Liste_AO()
        shows Liste_DI()
    Frame (0,430 800x50)
        shows Fusszeile_50()
END_VISUALIZATION

// VISUs/IBN/Liste_AO
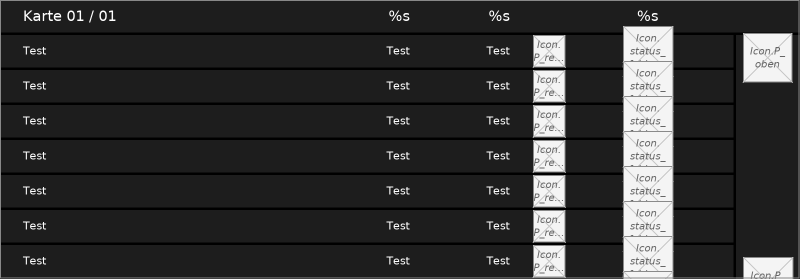
VISUALIZATION Liste_AO  // 800x279
    Rectangle (736,35 64x277)
    Image (743,257 50x50), image: Icon.P_unten
        OnMouseClick: execute {  }
    Image (743,33 49x49), image: Icon.P_oben
    Rectangle (0,35 733x32)
    Rectangle (20,35 400x32), "Test"
    Rectangle (0,105 733x32)
    Rectangle (20,105 400x32), "Test"
    Rectangle (0,70 733x32)
    Rectangle (20,70 400x32), "Test"
    Rectangle (0,140 733x32)
    Rectangle (20,140 400x32), "Test"
    Rectangle (0,210 733x32)
    Rectangle (20,210 400x32), "Test"
    Rectangle (0,175 733x32)
    Rectangle (20,175 400x32), "Test"
    Rectangle (0,420 733x32)
    Rectangle (20,420 400x32), "Test"
    Rectangle (0,245 733x32)
    Rectangle (20,245 400x32), "Test"
    Rectangle (0,315 733x32)
    Rectangle (20,315 400x32), "Test"
    Rectangle (0,280 733x32)
    Rectangle (20,280 400x32), "Test"
    Rectangle (0,350 733x32)
    Rectangle (20,350 400x32), "Test"
    Rectangle (0,385 733x32)
    Rectangle (20,385 400x32), "Test"
    Rectangle (0,0 800x32)
    Rectangle (20,0 324x32), "Karte 01 / 01"
    Rectangle (623,0 50x32), "%s", text list: 'Sprachen', text index: 49
    Group (333,26 340x50)
        Image (290,0 50x50), image: Icon.status_fehlerfrei_element
        Image (290,0 50x50), image: Icon.status_fehler_element
        Image (200,9 32x32), image: Icon.P_rechts
        Rectangle (100,9 80x32), "Test"
        Rectangle (0,9 80x32), "Test"
    Rectangle (433,0 80x32), "%s", text list: 'Sprachen', text index: 50
    Rectangle (333,0 80x32), "%s", text list: 'Sprachen', text index: 51
    Group (333,61 340x50)
        Image (290,0 50x50), image: Icon.status_fehlerfrei_element
        Image (290,0 50x50), image: Icon.status_fehler_element
        Image (200,9 32x32), image: Icon.P_rechts
        Rectangle (100,9 80x32), "Test"
        Rectangle (0,9 80x32), "Test"
    Group (333,96 340x50)
        Image (290,0 50x50), image: Icon.status_fehlerfrei_element
        Image (290,0 50x50), image: Icon.status_fehler_element
        Image (200,9 32x32), image: Icon.P_rechts
        Rectangle (100,9 80x32), "Test"
        Rectangle (0,9 80x32), "Test"
    Group (333,131 340x50)
        Image (290,0 50x50), image: Icon.status_fehlerfrei_element
        Image (290,0 50x50), image: Icon.status_fehler_element
        Image (200,9 32x32), image: Icon.P_rechts
        Rectangle (100,9 80x32), "Test"
        Rectangle (0,9 80x32), "Test"
    Group (333,166 340x50)
        Image (290,0 50x50), image: Icon.status_fehlerfrei_element
        Image (290,0 50x50), image: Icon.status_fehler_element
        Image (200,9 32x32), image: Icon.P_rechts
        Rectangle (100,9 80x32), "Test"
        Rectangle (0,9 80x32), "Test"
    Group (333,201 340x50)
        Image (290,0 50x50), image: Icon.status_fehlerfrei_element
        Image (290,0 50x50), image: Icon.status_fehler_element
        Image (200,9 32x32), image: Icon.P_rechts
        Rectangle (100,9 80x32), "Test"
        Rectangle (0,9 80x32), "Test"
    Group (333,236 340x50)
        Image (290,0 50x50), image: Icon.status_fehlerfrei_element
        Image (290,0 50x50), image: Icon.status_fehler_element
        Image (200,9 32x32), image: Icon.P_rechts
        Rectangle (100,9 80x32), "Test"
        Rectangle (0,9 80x32), "Test"
    Group (333,271 340x50)
        Image (290,0 50x50), image: Icon.status_fehlerfrei_element
        Image (290,0 50x50), image: Icon.status_fehler_element
        Image (200,9 32x32), image: Icon.P_rechts
        Rectangle (100,9 80x32), "Test"
        Rectangle (0,9 80x32), "Test"
    Group (333,306 340x50)
        Image (290,0 50x50), image: Icon.status_fehlerfrei_element
        Image (290,0 50x50), image: Icon.status_fehler_element
        Image (200,9 32x32), image: Icon.P_rechts
        Rectangle (100,9 80x32), "Test"
        Rectangle (0,9 80x32), "Test"
    Group (333,341 340x50)
        Image (290,0 50x50), image: Icon.status_fehlerfrei_element
        Image (290,0 50x50), image: Icon.status_fehler_element
        Image (200,9 32x32), image: Icon.P_rechts
        Rectangle (100,9 80x32), "Test"
        Rectangle (0,9 80x32), "Test"
    Group (333,376 340x50)
        Image (290,0 50x50), image: Icon.status_fehlerfrei_element
        Image (290,0 50x50), image: Icon.status_fehler_element
        Image (200,9 32x32), image: Icon.P_rechts
        Rectangle (100,9 80x32), "Test"
        Rectangle (0,9 80x32), "Test"
    Group (333,411 340x50)
        Image (290,0 50x50), image: Icon.status_fehlerfrei_element
        Image (290,0 50x50), image: Icon.status_fehler_element
        Image (200,9 32x32), image: Icon.P_rechts
        Rectangle (100,9 80x32), "Test"
        Rectangle (0,9 80x32), "Test"
END_VISUALIZATION

// VISUs/IBN/Liste_DI
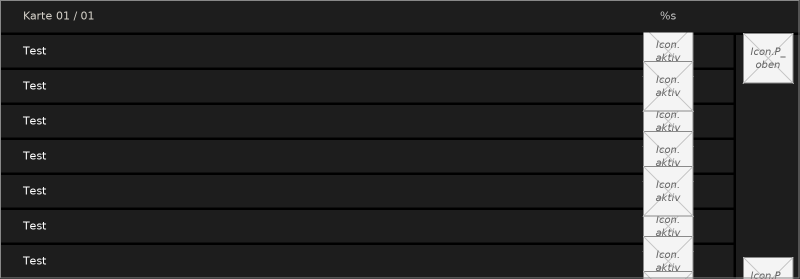
VISUALIZATION Liste_DI  // 800x279
    Rectangle (736,35 64x277)
    Image (743,257 50x50), image: Icon.P_unten
        OnMouseClick: execute {  }
    Image (743,33 50x50), image: Icon.P_oben
    Rectangle (0,35 733x32)
    Rectangle (0,105 733x32)
    Rectangle (0,70 733x32)
    Rectangle (0,140 733x32)
    Rectangle (0,210 733x32)
    Rectangle (0,175 733x32)
    Rectangle (0,420 733x32)
    Rectangle (0,245 733x32)
    Rectangle (0,315 733x32)
    Rectangle (0,280 733x32)
    Rectangle (0,350 733x32)
    Rectangle (0,385 733x32)
    Group (20,26 673x435)
        Rectangle (0,9 400x32), "Test"
        Image (623,0 50x50), image: Icon.inaktiv
        Image (623,0 50x50), image: Icon.aktiv
        Rectangle (0,79 400x32), "Test"
        Image (623,70 50x50), image: Icon.inaktiv
        Image (623,70 50x50), image: Icon.aktiv
        Rectangle (0,44 400x32), "Test"
        Image (623,35 50x50), image: Icon.inaktiv
        Image (623,35 50x50), image: Icon.aktiv
        Rectangle (0,114 400x32), "Test"
        Image (623,105 50x50), image: Icon.inaktiv
        Image (623,105 50x50), image: Icon.aktiv
        Rectangle (0,184 400x32), "Test"
        Image (623,175 50x50), image: Icon.inaktiv
        Image (623,175 50x50), image: Icon.aktiv
        Rectangle (0,149 400x32), "Test"
        Image (623,140 50x50), image: Icon.inaktiv
        Image (623,140 50x50), image: Icon.aktiv
        Rectangle (0,394 400x32), "Test"
        Image (623,385 50x50), image: Icon.inaktiv
        Image (623,385 50x50), image: Icon.aktiv
        Rectangle (0,219 400x32), "Test"
        Image (623,210 50x50), image: Icon.inaktiv
        Image (623,210 50x50), image: Icon.aktiv
        Rectangle (0,289 400x32), "Test"
        Image (623,280 50x50), image: Icon.inaktiv
        Image (623,280 50x50), image: Icon.aktiv
        Rectangle (0,254 400x32), "Test"
        Image (623,245 50x50), image: Icon.inaktiv
        Image (623,245 50x50), image: Icon.aktiv
        Rectangle (0,324 400x32), "Test"
        Image (623,315 50x50), image: Icon.inaktiv
        Image (623,315 50x50), image: Icon.aktiv
        Rectangle (0,359 400x32), "Test"
        Image (623,350 50x50), image: Icon.inaktiv
        Image (623,350 50x50), image: Icon.aktiv
    Group (0,0 800x32)
        Rectangle (0,0 800x32)
        Rectangle (20,0 324x32), "Karte 01 / 01"
        Rectangle (643,0 50x32), "%s", text list: 'Sprachen', text index: 49
END_VISUALIZATION

// VISUs/IBN/SW_IBN_Einstellungen_K
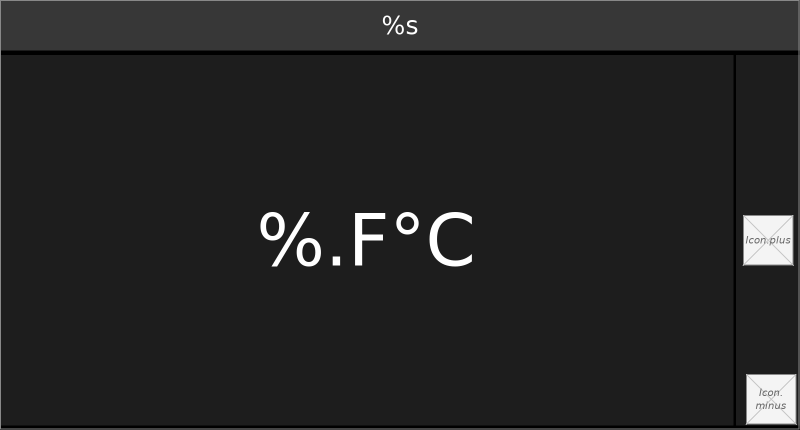
VISUALIZATION SW_IBN_Einstellungen_K  // 800x430
VAR_IN_OUT

END_VAR

VAR_INPUT
	i_titel:INT;
END_VAR
    Rectangle (0,0 800x50), "%s", text index: i_titel
    Rectangle (736,55 64x370)
    Image (743,215 50x50), image: Icon.plus
    Image (746,374 50x50), image: Icon.minus
    Rectangle (0,55 733x370), "%.F°C"
    Rectangle (401,485 150x30), "Zurück"
END_VISUALIZATION

// VISUs/Infoseite/Infoliste
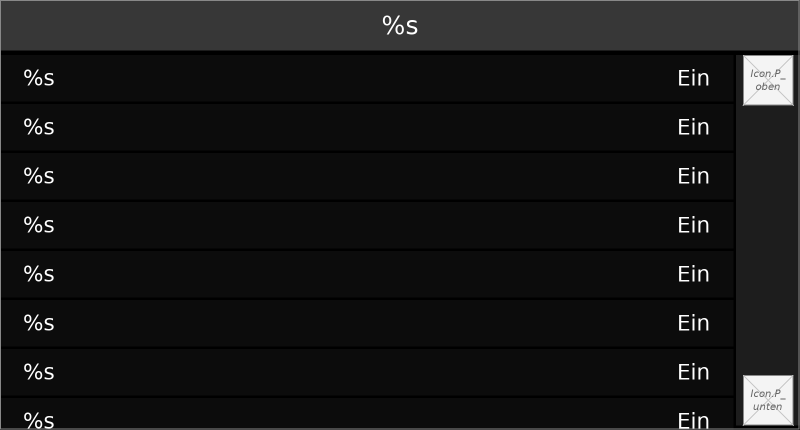
VISUALIZATION Infoliste  // 800x430
VAR_IN_OUT
	
END_VAR
VAR_INPUT
	i_Titel:INT;
	
END_VAR
VAR
	x_auf:BOOL;
	x_ab:BOOL;
	i_verschieben:INT:=0;
END_VAR
    Rectangle (0,0 800x50), "%s", text list: 'Sprachen', text index: i_Titel
    Rectangle (0,55 733x46)
    Label (20,55 479x46), "%s"
    Rectangle (0,104 733x46)
    Label (20,104 479x46), "%s"
    Rectangle (0,153 733x46)
    Label (20,153 479x46), "%s"
    Rectangle (0,202 733x46)
    Label (20,202 479x46), "%s"
    Rectangle (0,251 733x46)
    Label (20,251 479x46), "%s"
    Rectangle (0,300 733x46)
    Label (20,300 479x46), "%s"
    Rectangle (0,349 733x46)
    Label (20,349 479x46), "%s"
    Rectangle (583,55 130x46), "Ein"
    Rectangle (583,104 130x46), "Ein"
    Rectangle (0,398 733x46)
    Label (20,398 479x46), "%s"
    Rectangle (0,447 733x46)
    Label (20,447 479x46), "%s"
    Rectangle (0,496 733x46)
    Label (20,496 479x46), "%s"
    Rectangle (0,545 733x46)
    Label (20,545 479x46), "%s"
    Rectangle (583,545 130x46), "Ein"
    Rectangle (0,594 733x46)
    Label (20,594 479x46), "%s"
    Rectangle (583,153 130x46), "Ein"
    Rectangle (583,202 130x46), "Ein"
    Rectangle (583,251 130x46), "Ein"
    Rectangle (583,349 130x46), "Ein"
    Rectangle (583,300 130x46), "Ein"
    Rectangle (583,398 130x46), "Ein"
    Rectangle (583,447 130x46), "Ein"
    Rectangle (583,496 130x46), "Ein"
    Rectangle (583,594 130x46), "Ein"
    Group (736,55 64x370)
        Rectangle (0,0 64x370)
        Image (7,320 50x50), image: Icon.P_unten
            OnMouseClick:  ToggleVariable=x_ab
            OnMouseClick: execute {
                IF x_ab THEN
                	i_verschieben:=i_verschieben+50;
                	x_ab:=0;
                END_IF
            }
        Image (7,0 50x50), image: Icon.P_oben
            OnMouseClick:  ToggleVariable=x_auf
            OnMouseClick: execute {
                IF x_auf THEN
                	i_verschieben:=i_verschieben-50;
                	x_auf:=0;
                END_IF
            }
END_VISUALIZATION

// VISUs/Infoseite/Infoseite
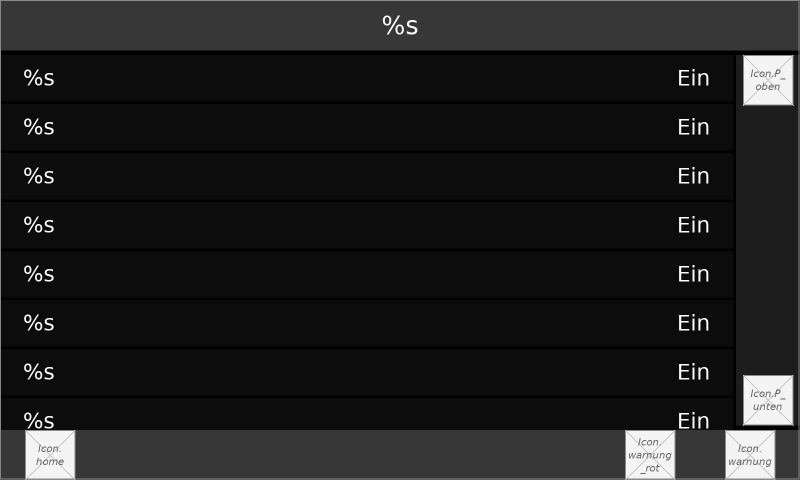
VISUALIZATION Infoseite  // 800x480
    Frame (0,0 800x430)
        shows Infoliste(i_Titel := 31)
    Frame (0,430 800x50)
        shows Fusszeile_50()
END_VISUALIZATION

// VISUs/Sollwertmenu_9/Sollwertmenu/Sollwertmenu
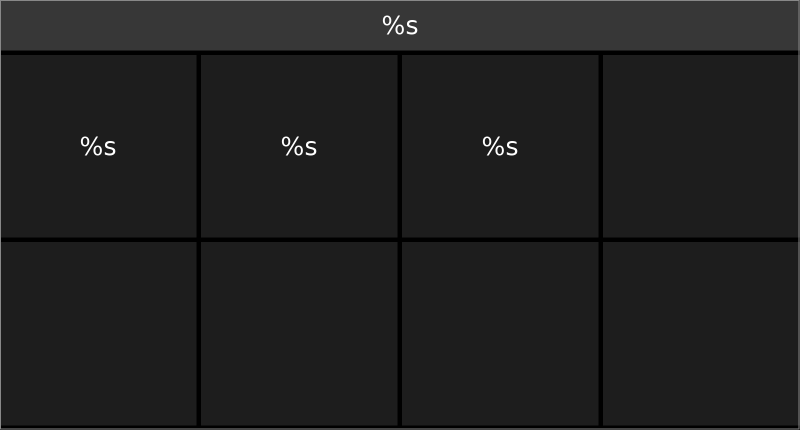
VISUALIZATION Sollwertmenu  // 800x430
    Rectangle (0,0 800x50), "%s", text list: 'Sprachen', text index: 3
    Rectangle (0,55 196x182), "%s", text list: 'Sprachen', text index: 0
        OnMouseClick:  Assign=Sollwertmenu_Waermegewinnung, Type=Assignment
    Rectangle (201,55 196x182), "%s", text list: 'Sprachen', text index: 1
        OnMouseClick:  Assign=Sollwertmenu_Waermepumpe, Type=Assignment
    Rectangle (402,55 196x182), "%s", text list: 'Sprachen', text index: 2
        OnMouseClick:  Assign=Sollwertmenu_Waermesenke, Type=Assignment
    Rectangle (603,55 197x182)
    Rectangle (0,242 196x183)
    Rectangle (201,242 196x183)
    Rectangle (402,242 196x183)
    Rectangle (603,242 197x183)
    Frame (0,430 800x50)
        shows Fusszeile_50()
    Image (125,430 50x50), image: Icon.zurueck
        OnMouseClick:  Assign=Hauptmenu, Type=Assignment
END_VISUALIZATION

// VISUs/Sollwertmenu_9/Wärmegewinnung/UWP/SW_Einstellungen_C
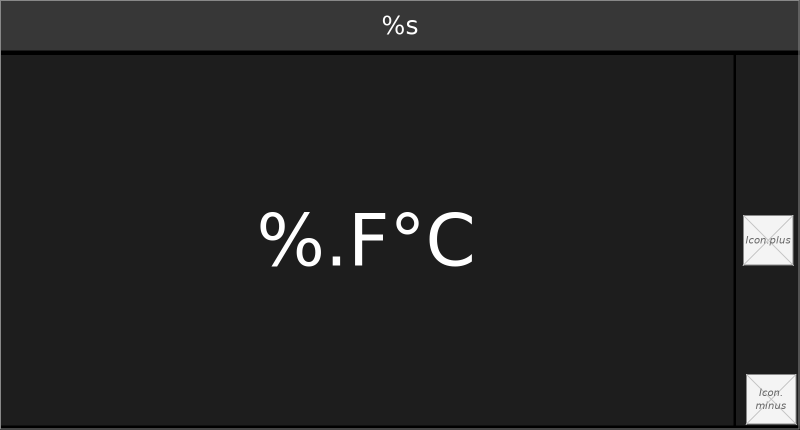
VISUALIZATION SW_Einstellungen_C  // 800x430
VAR_IN_OUT
		
END_VAR

VAR_INPUT
	i_titel:INT;
END_VAR
    Rectangle (0,0 800x50), "%s", text list: 'Sprachen', text index: i_titel
    Rectangle (736,55 64x370)
    Image (743,215 50x50), image: Icon.plus
    Image (746,374 50x50), image: Icon.minus
    Rectangle (0,55 733x370), "%.F°C"
    Rectangle (401,485 150x30), "Zurück"
        OnMouseClick: execute { GWP_Library.Visu.i_Frame_Index:=0; }
        OnMouseClick: FrameSelectionChange Selection=Selection=-1, GlobSel=AssignDir=Test_SW_WP.GenElemInst_5, AssignType=Directly, SelType=Globally
END_VISUALIZATION

// VISUs/Sollwertmenu_9/Wärmegewinnung/UWP/SW_Einstellungen_DT
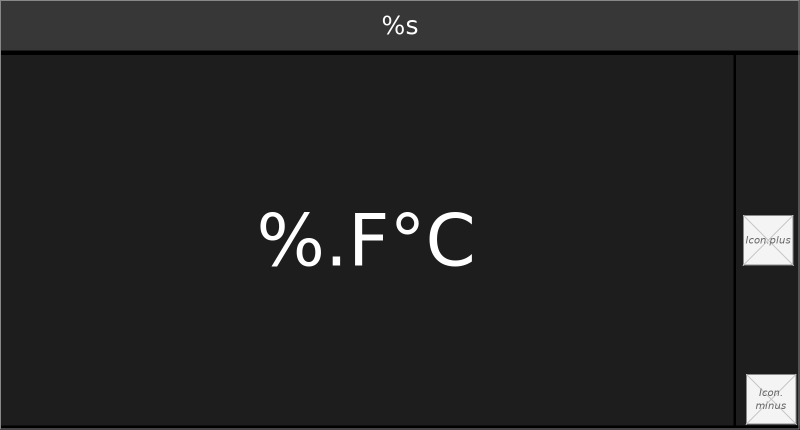
VISUALIZATION SW_Einstellungen_DT  // 800x430
VAR_IN_OUT
		
END_VAR

VAR_INPUT
	i_titel:INT;
END_VAR
    Rectangle (0,0 800x50), "%s", text list: 'Sprachen', text index: i_titel
    Rectangle (736,55 64x370)
    Image (743,215 50x50), image: Icon.plus
    Image (746,374 50x50), image: Icon.minus
    Rectangle (0,55 733x370), "%.F°C"
    Rectangle (401,485 150x30), "Zurück"
        OnMouseClick: execute { GWP_Library.Visu.i_Frame_Index:=0; }
        OnMouseClick: FrameSelectionChange Selection=Selection=-1, GlobSel=AssignDir=Test_SW_WP.GenElemInst_5, AssignType=Directly, SelType=Globally
END_VISUALIZATION

// VISUs/Sollwertmenu_9/Wärmegewinnung/UWP/SW_Einstellungen_K
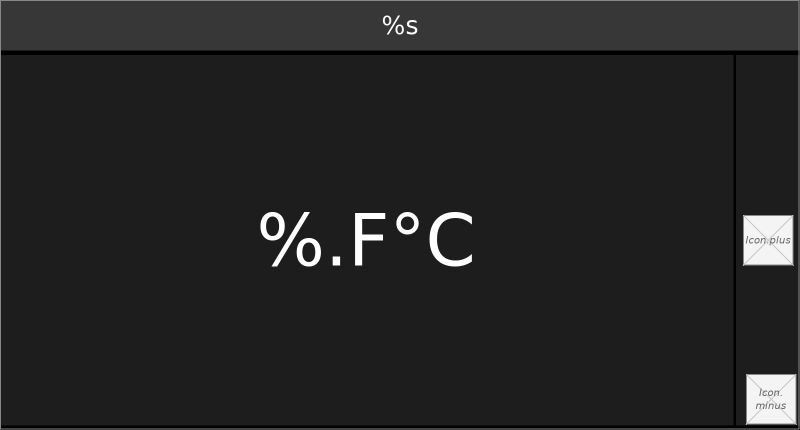
VISUALIZATION SW_Einstellungen_K  // 800x430
VAR_IN_OUT

END_VAR

VAR_INPUT
	i_titel:INT;
END_VAR
    Rectangle (0,0 800x50), "%s", text index: i_titel
    Rectangle (736,55 64x370)
    Image (743,215 50x50), image: Icon.plus
    Image (746,374 50x50), image: Icon.minus
    Rectangle (0,55 733x370), "%.F°C"
    Rectangle (401,485 150x30), "Zurück"
        OnMouseClick: execute { GWP_Library.Visu.i_Frame_Index:=0; }
        OnMouseClick: FrameSelectionChange Selection=Selection=-1, GlobSel=AssignDir=Test_SW_WP.GenElemInst_5, AssignType=Directly, SelType=Globally
END_VISUALIZATION

// VISUs/Sollwertmenu_9/Wärmegewinnung/UWP/SW_Einstellungen_Zeit
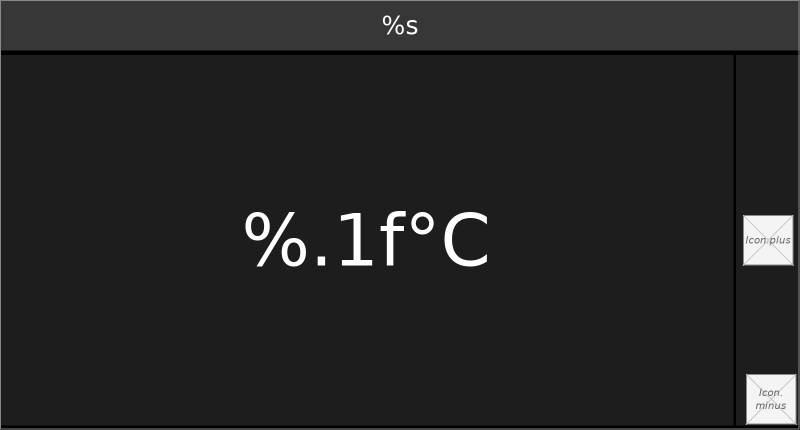
VISUALIZATION SW_Einstellungen_Zeit  // 800x430
VAR_IN_OUT
	f_Data:REAL;
	
END_VAR

VAR_INPUT
	i_titel:INT;
END_VAR

VAR
	Timer:ton;
END_VAR
    Rectangle (0,0 800x50), "%s", text list: 'Sprachen', text index: i_titel
    Rectangle (736,55 64x370)
    Image (743,215 50x50), image: Icon.plus
        OnMouseClick: execute { f_data:=f_data + 1; }
    Image (746,374 50x50), image: Icon.minus
        OnMouseClick: execute { f_data:=f_data - 1; }
    Rectangle (0,55 733x370), "%.1f°C", text variable: f_Data
    Image (836,328 50x50), image: Icon.zurueck
        OnMouseClick: execute { GWP_Library.Visu.i_Frame_Index:=0; }
END_VISUALIZATION

// VISUs/Sollwertmenu_9/Wärmegewinnung/UWP/SW_WG_UWP_Verd
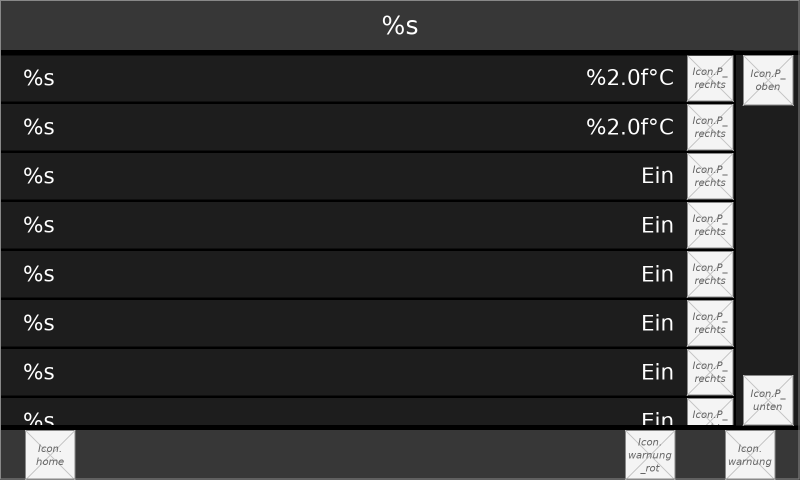
VISUALIZATION SW_WG_UWP_Verd  // 800x480
VAR_IN_OUT
	FB_GR2:GR_2;
END_VAR
    Frame (0,0 800x430), frame switch variable: GWP_Library.Visu.i_Frame_Index
        shows SW_WG_UWP_Verd_Liste(i_Titel := 25, FB_GR2 := FB_GR2)
        shows SW_Einstellungen_Zeit(i_titel := 30, f_Data := FB_GR2.f_AT)
        shows SW_Einstellungen_DT()
        shows SW_Einstellungen_K()
        shows SW_Einstellungen_Zeit(i_titel := 30)
    Frame (0,430 800x50)
        shows Fusszeile_50()
END_VISUALIZATION

// VISUs/Sollwertmenu_9/Wärmegewinnung/UWP/SW_WG_UWP_Verd_Liste
